(* IEC 61131-3 sources: ecmc_strucpp_app_example/ioc_project_example/src, 3 files *)

(* ---- main_counter_fb.st ---- *)
FUNCTION_BLOCK COUNTER_FB
VAR_INPUT
  Enable : BOOL;
END_VAR
VAR_OUTPUT
  Value : INT;
END_VAR

IF Enable THEN
  Value := Value + 1;
ELSE
  Value := 0;
END_IF;
END_FUNCTION_BLOCK

(* ---- machine.st ---- *)
PROGRAM MACHINE
VAR
  start_button   AT %IX0.0 : BOOL;  // @ecmc ec0.s2.mm.inputDataArray01
  stop_button    AT %IX0.1 : BOOL;  // @ecmc ec0.s2.mm.inputDataArray01
  enable_output  AT %QX0.0 : BOOL;  // @ecmc ec0.s2.mm.outputDataArray01
  target_word    AT %QW2   : INT;   // @ecmc ec0.s2.mm.outputDataArray01
  counter        AT %MW0   : INT;   // @epics plugin.strucpp.machine.counter
  manual_target            : INT;   // @epics plugin.strucpp.machine.manual_target rw
  counter_fb               : COUNTER_FB;
END_VAR

IF stop_button THEN
  enable_output := FALSE;
ELSIF start_button THEN
  enable_output := TRUE;
END_IF;

counter_fb(Enable := enable_output);
counter := counter_fb.Value;

IF enable_output THEN
  IF manual_target <> 0 THEN
    target_word := manual_target;
  ELSE
    target_word := counter;
  END_IF;
ELSE
  target_word := 0;
END_IF;
END_PROGRAM

(* ---- main.st ---- *)
PROGRAM MAIN
VAR
  actual_position    AT %IW0 : INT;   // @ecmc ec0.s14.positionActual01
  drive_control      AT %QW0 : WORD;  // @ecmc ec0.s14.driveControl01
  velocity_setpoint  AT %QW2 : INT;   // @ecmc ec0.s14.velocitySetpoint01
  cycle_counter      AT %MW0 : INT;   // @epics
  manual_velocity             : INT;   // @epics rw
  actual_pos_export           : INT;   // @epics
  counter_fb                  : COUNTER_FB;
END_VAR

actual_pos_export := actual_position;
drive_control := 16#0001;
counter_fb(Enable := TRUE);
cycle_counter := counter_fb.Value;

IF manual_velocity <> 0 THEN
  velocity_setpoint := manual_velocity;
ELSIF actual_position < 1000 THEN
  velocity_setpoint := 1000;
ELSE
  velocity_setpoint := -1000;
END_IF;
END_PROGRAM
